// TIA Portal V16 export
// export: Created 2021-07-03T21:22:41.7291853Z, ExportSetting WithDefaults, DisplayName Totally Integrated Automation Portal, DisplayVersion V16, DisplayName TIA Portal Version Control Interface, DisplayVersion V16, DisplayName TIA Portal Openness, DisplayVersion V16, DisplayName STEP 7 Professional, DisplayVersion V16, DisplayName STEP 7 Safety, DisplayVersion V16, DisplayName WinCC Professional, DisplayVersion V16
DATA_BLOCK "Data"   // DB4
{ S7_Optimized_Access := 'FALSE'; DB_Accessible_From_OPC_UA := 'FALSE' }
VERSION : 0.1
// stored: AutoNumber true, DBAccessibleFromOPCUA false, IsOnlyStoredInLoadMemory false, IsWriteProtectedInAS false
   VAR
      Receive { ExternalAccessible := 'False'; ExternalVisible := 'False'; ExternalWritable := 'False'} : Array[0..99] of Byte;
      Send { ExternalAccessible := 'False'; ExternalVisible := 'False'; ExternalWritable := 'False'} : Array[0..99] of Byte;
   END_VAR
BEGIN
   Send[0..1] := 16#A;
   Send[2..3] := 16#B;
   Send[4..5] := 16#C;
   Send[6..7] := 16#D;
   Send[8..9] := 16#E;
   Send[10..11] := 16#F;
   Send[12] := 11;
   Send[13] := 12;
   Send[14] := 13;
   Send[15] := 14;
   Send[16] := 15;
   Send[17] := 16;
   Send[18] := 17;
   Send[19] := 18;
   Send[20] := 19;
   Send[99] := 16#FF;
END_DATA_BLOCK
